// SIMATIC S7-200 project (STEP 7-Micro/WIN), CPU 224XP REL 02.01

SYMBOL_TABLE USUARIO1
FC_1_SILO_1      I0.0
FC_2_SILO1       I0.1
FC_3_SILO2       I0.2
FC_4_SILO2       I0.3
TOLVA            Q0.0
TORNILLO_SIN_FIN Q0.1
COMPUERTA_1      Q0.2
CINTA_1          Q0.3
COMPUERTA_2      Q0.4
CINTA_5          Q0.5
END_SYMBOL_TABLE

ORGANIZATION_BLOCK PRINCIPAL:OB1
TITLE=COMENTARIOS DEL PROGRAMA
BEGIN
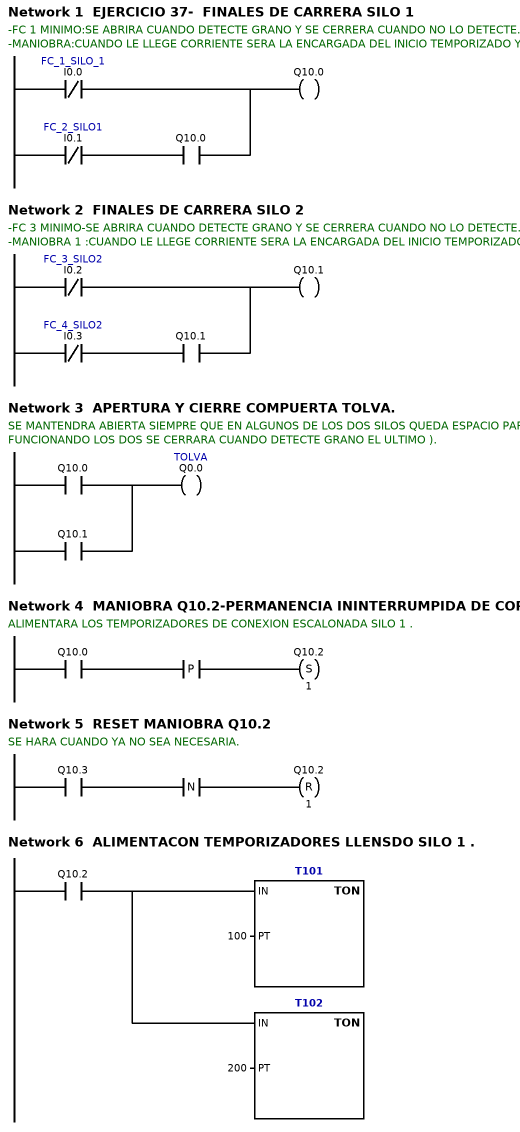
Network 1 // EJERCICIO 37-  FINALES DE CARRERA SILO 1 

// -FC 1 MINIMO:SE ABRIRA CUANDO DETECTE GRANO Y SE CERRERA CUANDO NO LO DETECTE.
// -FC 2 MAXIMO:"        "              "                  "           "        "  "         "                 "          "     "         "  
// -MANIOBRA:CUANDO LE LLEGE CORRIENTE SERA LA ENCARGADA DEL INICIO TEMPORIZADO Y CUANDO DEJE DE LLEGARLE INICIARA LA SECUENCIA TEMPORIZADA DE DESCONEXION.
LDN    FC_1_SILO_1:I0.0
LDN    FC_2_SILO1:I0.1
A      Q10.0
OLD
=      Q10.0
Network 2 // FINALES DE CARRERA SILO 2 
// -FC 3 MINIMO-SE ABRIRA CUANDO DETECTE GRANO Y SE CERRERA CUANDO NO LO DETECTE.
// -FC 4 MAXIMO:"        "                 "            "              "        "  "           "               "           "   "         2
// -MANIOBRA 1 :CUANDO LE LLEGE CORRIENTE SERA LA ENCARGADA DEL INICIO TEMPORIZADO Y CUANDO DEJE DE LLEGARLE INICIARA LA SECUENCIA TEMPORIZADA DE DESCONEXION.
LDN    FC_3_SILO2:I0.2
LDN    FC_4_SILO2:I0.3
A      Q10.1
OLD
=      Q10.1
Network 3 // APERTURA Y CIERRE COMPUERTA TOLVA.
// SE MANTENDRA ABIERTA SIEMPRE QUE EN ALGUNOS DE LOS DOS SILOS QUEDA ESPACIO PARA EL GRANO.CUANDO LOS FC MAXIMO DETECTEN GRANO SE CERRARA(SIEMPRE QUE ESTEN FUNCIONANDO LOS DOS SE CERRARA CUANDO DETECTE GRANO EL ULTIMO ).
LD     Q10.0
O      Q10.1
=      TOLVA:Q0.0
Network 4 // MANIOBRA Q10.2-PERMANENCIA ININTERRUMPIDA DE CORRIENTE SILO 1.
// ALIMENTARA LOS TEMPORIZADORES DE CONEXION ESCALONADA SILO 1 .
LD     Q10.0
EU
S      Q10.2, 1
Network 5 // RESET MANIOBRA Q10.2
// SE HARA CUANDO YA NO SEA NECESARIA.
LD     Q10.3
ED
R      Q10.2, 1
Network 6 // ALIMENTACON TEMPORIZADORES LLENSDO SILO 1 .
LD     Q10.2
TON    T101, 100
TON    T102, 200
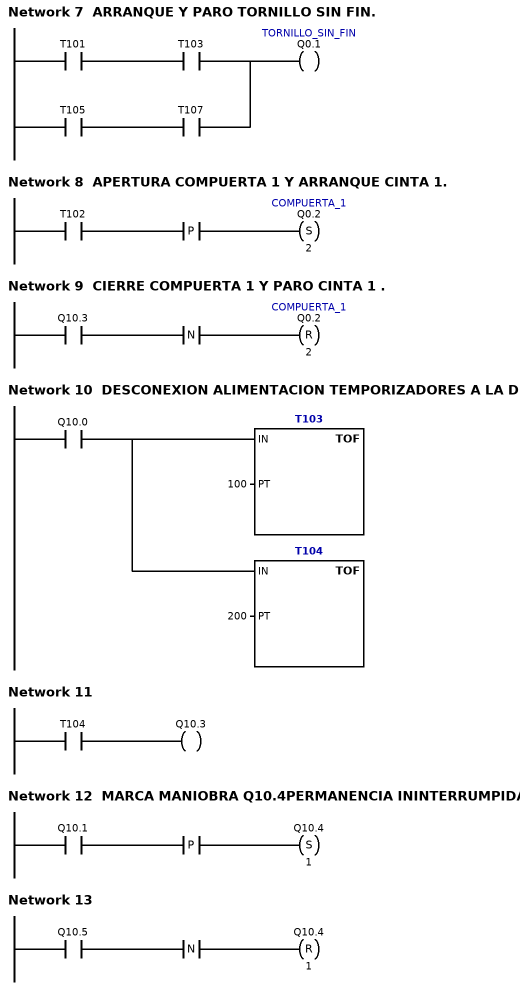
Network 7 // ARRANQUE Y PARO TORNILLO SIN FIN.
LD     T101
A      T103
LD     T105
A      T107
OLD
=      TORNILLO_SIN_FIN:Q0.1
Network 8 // APERTURA COMPUERTA 1 Y ARRANQUE CINTA 1.
LD     T102
EU
S      COMPUERTA_1:Q0.2, 2
Network 9 // CIERRE COMPUERTA 1 Y PARO CINTA 1 .
LD     Q10.3
ED
R      COMPUERTA_1:Q0.2, 2
Network 10 // DESCONEXION ALIMENTACION TEMPORIZADORES A LA DESCONEXION.
LD     Q10.0
TOF    T103, 100
TOF    T104, 200
Network 11
LD     T104
=      Q10.3
Network 12 // MARCA MANIOBRA Q10.4PERMANENCIA ININTERRUMPIDA DE CORRIENTE SILO 2.
LD     Q10.1
EU
S      Q10.4, 1
Network 13
LD     Q10.5
ED
R      Q10.4, 1
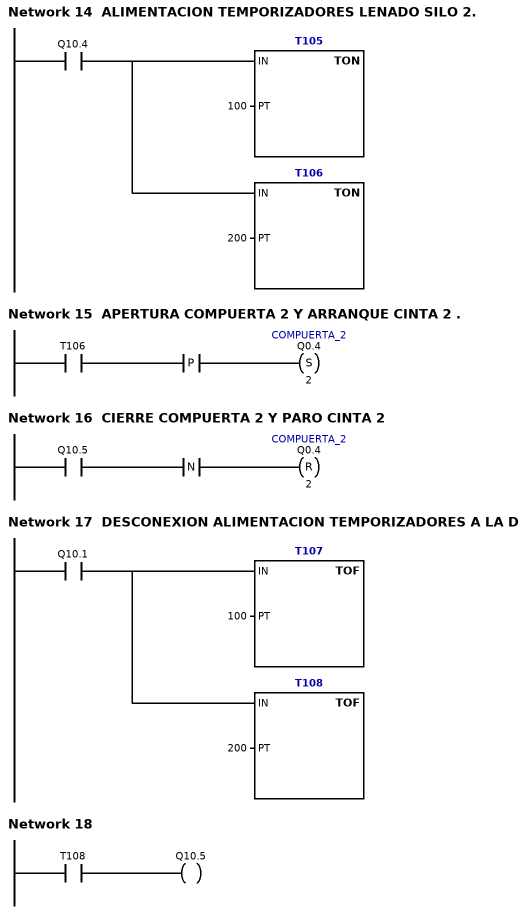
Network 14 // ALIMENTACION TEMPORIZADORES LENADO SILO 2.
LD     Q10.4
TON    T105, 100
TON    T106, 200
Network 15 // APERTURA COMPUERTA 2 Y ARRANQUE CINTA 2 .
LD     T106
EU
S      COMPUERTA_2:Q0.4, 2
Network 16 // CIERRE COMPUERTA 2 Y PARO CINTA 2 
LD     Q10.5
ED
R      COMPUERTA_2:Q0.4, 2
Network 17 // DESCONEXION ALIMENTACION TEMPORIZADORES A LA DESCONEXION.
LD     Q10.1
TOF    T107, 100
TOF    T108, 200
Network 18
LD     T108
=      Q10.5
END_ORGANIZATION_BLOCK
